{attribute 'hide'}
INTERFACE INTERNAL IStringBuilder

METHOD Append : IStringBuilder // Append text TO t current build STRING.
VAR_INPUT
    Text : Tc2_System.T_MaxString; //Text to append to current build string
END_VAR
END_METHOD

METHOD AppendIf : IStringBuilder
VAR_INPUT
    Condition : BOOL;
    Text : Tc2_System.T_MaxString;
END_VAR
END_METHOD

METHOD InsertAtLocation : IStringBuilder
VAR_INPUT
    Text : Tc2_System.T_MaxString;
    Position : INT;
END_VAR
END_METHOD

METHOD PadLeft : IStringBuilder
VAR_INPUT
    Text : Tc2_System.T_MaxString; // Text to append to current build string
    Length : INT; // Total length of text + padding
    Char : STRING(1); // Character to be padded left of text
END_VAR
END_METHOD

METHOD Reset : ILimitedStringBuilder //Reset current build STRING TO an empty STRING.
END_METHOD

METHOD ToString : Tc2_System.T_MaxString //Returns current build STRING.
END_METHOD

END_INTERFACE

(* stored: Version 1.1.0.1, ProductVersion 3.1.4024.12
   Itf IStringBuilder: Id {cc6d396c-ab11-4512-b217-fcaa420ac27e}
   Method Append: Id {39f6182f-ddaa-4a04-88e3-b41671a4f64d}
   Method AppendIf: Id {04ce72ab-2dd5-4f0f-9870-b897f32c1a5a}
   Method InsertAtLocation: Id {84b072e0-2852-4c7d-a45f-8bbe495344a7}
   Method PadLeft: Id {c4fcdbc5-50e6-479f-bc91-2aff2727bcfd}
   Method Reset: Id {6ef3d071-ad38-492e-ac0f-193eb38816d5}
   Method ToString: Id {857ec4df-c977-46b4-ad47-ee4fdd52fb44} *)
